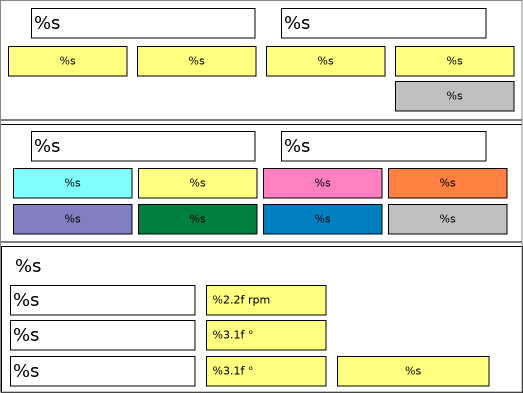
VISUALIZATION VISU_AXE_STD1_LIN_ROT_FCT_CONS_OSC  // 523x393
VAR_IN_OUT
	m_Input_MOTEUR: BLOCK_AXE_STD1_OSCILLANT;
	m_Input_PRG_MOUVEMENT_PS: BLOCK_PRG_MOUVEMENT_PS;
END_VAR
VAR_INPUT CONSTANT
	m_Input_INDEX_MOTEUR : INT;
END_VAR
    Rectangle (0,0 522x120)
    RoundedRectangle (31,8 224x30), "%s", text list: 'TextList_Moteurs', text index: 13
    RoundedRectangle (281,8 205x30), "%s", text variable: m_Input_MOTEUR.CONF_ID_Poste[m_Input_MOTEUR.PRM_NPoste]
    RoundedRectangle (8,46 119x30), "%s", text variable: m_Input_MOTEUR.CONF_ID_Poste[1], invisible if: m_Input_PRG_MOUVEMENT_PS.CONF_NB_POSTE[m_Input_INDEX_MOTEUR]<1, input disabled if: (NOT PRG_User.ACTU_USER.MAINTENANCE AND m_Input_MOTEUR.MANUAL) OR (NOT PRG_User.ACTU_USER.FONCTION_SA AND NOT m_Input_MOTEUR.MANUAL)
        OnMouseClick: execute { m_Input_MOTEUR.PRM_NPOSTE:=1; }
    RoundedRectangle (395,81 119x30), "%s", text variable: m_Input_MOTEUR.CONF_ID_POSTE[0], invisible if: NOT m_Input_PRG_MOUVEMENT_PS.CONF_Use_Poste0[m_Input_INDEX_MOTEUR], input disabled if: (NOT PRG_User.ACTU_USER.MAINTENANCE AND m_Input_MOTEUR.MANUAL) OR (NOT PRG_User.ACTU_USER.FONCTION_SA AND NOT m_Input_MOTEUR.MANUAL)
        OnMouseClick: execute { m_Input_MOTEUR.PRM_NPOSTE:=0; }
    RoundedRectangle (137,46 119x30), "%s", text variable: m_Input_MOTEUR.CONF_ID_Poste[2], invisible if: m_Input_PRG_MOUVEMENT_PS.CONF_NB_POSTE[m_Input_INDEX_MOTEUR]<2, input disabled if: (NOT PRG_User.ACTU_USER.MAINTENANCE AND m_Input_MOTEUR.MANUAL) OR (NOT PRG_User.ACTU_USER.FONCTION_SA AND NOT m_Input_MOTEUR.MANUAL)
        OnMouseClick: execute { m_Input_MOTEUR.PRM_NPOSTE:=2; }
    RoundedRectangle (266,46 119x30), "%s", text variable: m_Input_MOTEUR.CONF_ID_Poste[3], invisible if: m_Input_PRG_MOUVEMENT_PS.CONF_NB_POSTE[m_Input_INDEX_MOTEUR]<3, input disabled if: (NOT PRG_User.ACTU_USER.MAINTENANCE AND m_Input_MOTEUR.MANUAL) OR (NOT PRG_User.ACTU_USER.FONCTION_SA AND NOT m_Input_MOTEUR.MANUAL)
        OnMouseClick: execute { m_Input_MOTEUR.PRM_NPOSTE:=3; }
    RoundedRectangle (395,46 119x30), "%s", text variable: m_Input_MOTEUR.CONF_ID_Poste[4], invisible if: m_Input_PRG_MOUVEMENT_PS.CONF_NB_POSTE[m_Input_INDEX_MOTEUR]<4, input disabled if: (NOT PRG_User.ACTU_USER.MAINTENANCE AND m_Input_MOTEUR.MANUAL) OR (NOT PRG_User.ACTU_USER.FONCTION_SA AND NOT m_Input_MOTEUR.MANUAL)
        OnMouseClick: execute { m_Input_MOTEUR.PRM_NPOSTE:=4; }
    Rectangle (0,124 522x118)
    RoundedRectangle (31,131 224x30), "%s", text list: 'TextList_Moteurs', text index: 14
    RoundedRectangle (281,131 205x30), "%s", text variable: m_Input_MOTEUR.CONF_ID_Ref[m_Input_MOTEUR.PRM_NRef]
    RoundedRectangle (13,168 119x30), "%s", text variable: m_Input_MOTEUR.CONF_ID_REF[1], invisible if: m_Input_PRG_MOUVEMENT_PS.CONF_NB_REF[m_Input_INDEX_MOTEUR]<1, input disabled if: (NOT PRG_User.ACTU_USER.MAINTENANCE AND m_Input_MOTEUR.MANUAL) OR (NOT PRG_User.ACTU_USER.FONCTION_SA AND NOT m_Input_MOTEUR.MANUAL)
        OnMouseClick: execute { m_Input_MOTEUR.PRM_NREF:=1; }
    RoundedRectangle (138,168 119x30), "%s", text variable: m_Input_MOTEUR.CONF_ID_REF[2], invisible if: m_Input_PRG_MOUVEMENT_PS.CONF_NB_REF[m_Input_INDEX_MOTEUR]<2, input disabled if: (NOT PRG_User.ACTU_USER.MAINTENANCE AND m_Input_MOTEUR.MANUAL) OR (NOT PRG_User.ACTU_USER.FONCTION_SA AND NOT m_Input_MOTEUR.MANUAL)
        OnMouseClick: execute { m_Input_MOTEUR.PRM_NREF:=2; }
    RoundedRectangle (263,168 119x30), "%s", text variable: m_Input_MOTEUR.CONF_ID_REF[3], invisible if: m_Input_PRG_MOUVEMENT_PS.CONF_NB_REF[m_Input_INDEX_MOTEUR]<3, input disabled if: (NOT PRG_User.ACTU_USER.MAINTENANCE AND m_Input_MOTEUR.MANUAL) OR (NOT PRG_User.ACTU_USER.FONCTION_SA AND NOT m_Input_MOTEUR.MANUAL)
        OnMouseUp: execute { m_Input_MOTEUR.PRM_NREF:=3; }
    RoundedRectangle (388,168 119x30), "%s", text variable: m_Input_MOTEUR.CONF_ID_REF[4], invisible if: m_Input_PRG_MOUVEMENT_PS.CONF_NB_REF[m_Input_INDEX_MOTEUR]<4, input disabled if: (NOT PRG_User.ACTU_USER.MAINTENANCE AND m_Input_MOTEUR.MANUAL) OR (NOT PRG_User.ACTU_USER.FONCTION_SA AND NOT m_Input_MOTEUR.MANUAL)
        OnMouseClick: execute { m_Input_MOTEUR.PRM_NREF:=4; }
    RoundedRectangle (13,204 119x30), "%s", text variable: m_Input_MOTEUR.CONF_ID_REF[5], invisible if: m_Input_PRG_MOUVEMENT_PS.CONF_NB_REF[m_Input_INDEX_MOTEUR]<5, input disabled if: (NOT PRG_User.ACTU_USER.MAINTENANCE AND m_Input_MOTEUR.MANUAL) OR (NOT PRG_User.ACTU_USER.FONCTION_SA AND NOT m_Input_MOTEUR.MANUAL)
        OnMouseClick: execute { m_Input_MOTEUR.PRM_NREF:=5; }
    RoundedRectangle (138,204 119x30), "%s", text variable: m_Input_MOTEUR.CONF_ID_REF[6], invisible if: m_Input_PRG_MOUVEMENT_PS.CONF_NB_REF[m_Input_INDEX_MOTEUR]<6, input disabled if: (NOT PRG_User.ACTU_USER.MAINTENANCE AND m_Input_MOTEUR.MANUAL) OR (NOT PRG_User.ACTU_USER.FONCTION_SA AND NOT m_Input_MOTEUR.MANUAL)
        OnMouseClick: execute { m_Input_MOTEUR.PRM_NREF:=6; }
    RoundedRectangle (388,204 119x30), "%s", text variable: m_Input_MOTEUR.CONF_ID_REF[0], invisible if: NOT m_Input_PRG_MOUVEMENT_PS.CONF_Use_Ref0[m_Input_INDEX_MOTEUR], input disabled if: (NOT PRG_User.ACTU_USER.MAINTENANCE AND m_Input_MOTEUR.MANUAL) OR (NOT PRG_User.ACTU_USER.FONCTION_SA AND NOT m_Input_MOTEUR.MANUAL)
        OnMouseClick: execute { m_Input_MOTEUR.PRM_NREF:=0; }
    RoundedRectangle (263,204 119x30), "%s", text variable: m_Input_MOTEUR.CONF_ID_REF[7], invisible if: m_Input_PRG_MOUVEMENT_PS.CONF_NB_REF[m_Input_INDEX_MOTEUR]<7, input disabled if: (NOT PRG_User.ACTU_USER.MAINTENANCE AND m_Input_MOTEUR.MANUAL) OR (NOT PRG_User.ACTU_USER.FONCTION_SA AND NOT m_Input_MOTEUR.MANUAL)
        OnMouseClick: execute { m_Input_MOTEUR.PRM_NREF:=7; }
    Rectangle (1,246 522x147)
    RoundedRectangle (10,320 185x30), "%s", invisible if: NOT m_Input_PRG_MOUVEMENT_PS.CONF_Balayage[m_Input_INDEX_MOTEUR] AND NOT m_Input_PRG_MOUVEMENT_PS.CONF_Positionnement[m_Input_INDEX_MOTEUR], text list: 'TextList_Moteurs', text index: 12
    RoundedRectangle (206,320 120x30), "%3.1f mm", text variable: m_Input_MOTEUR.PRM_Position, invisible if: (NOT m_Input_PRG_MOUVEMENT_PS.CONF_Balayage[m_Input_INDEX_MOTEUR] AND NOT m_Input_PRG_MOUVEMENT_PS.CONF_Positionnement[m_Input_INDEX_MOTEUR]) OR NOT m_Input_MOTEUR.CONF_Mvt_Lineaire, input disabled if: (NOT PRG_User.ACTU_USER.MAINTENANCE AND m_Input_MOTEUR.MANUAL) OR (NOT PRG_User.ACTU_USER.FONCTION_SA AND NOT m_Input_MOTEUR.MANUAL)
        OnMouseClick: write the text variable via VisuDialogs.Numpad, min m_Input_PRG_MOUVEMENT_PS.CONF_MIN_POS[m_Input_INDEX_MOTEUR], max m_Input_PRG_MOUVEMENT_PS.CONF_MAX_POS[m_Input_INDEX_MOTEUR]
    RoundedRectangle (10,285 185x30), "%s", invisible if: NOT m_Input_PRG_MOUVEMENT_PS.CONF_Balayage[m_Input_INDEX_MOTEUR] AND NOT m_Input_PRG_MOUVEMENT_PS.CONF_Rotation[m_Input_INDEX_MOTEUR], text list: 'TextList_Moteurs', text index: 7
    RoundedRectangle (206,285 120x30), "%2.2f mmps", text variable: m_Input_MOTEUR.PRM_V_BalRot, invisible if: (NOT m_Input_PRG_MOUVEMENT_PS.CONF_Balayage[m_Input_INDEX_MOTEUR] AND NOT m_Input_PRG_MOUVEMENT_PS.CONF_Rotation[m_Input_INDEX_MOTEUR]) OR NOT m_Input_MOTEUR.CONF_Mvt_Lineaire, input disabled if: (NOT PRG_User.ACTU_USER.MAINTENANCE AND m_Input_MOTEUR.MANUAL) OR (NOT PRG_User.ACTU_USER.FONCTION_SA AND NOT m_Input_MOTEUR.MANUAL)
        OnMouseClick: write the text variable via VisuDialogs.Numpad, min m_Input_PRG_MOUVEMENT_PS.CONF_MIN_SPEED[m_Input_INDEX_MOTEUR], max m_Input_PRG_MOUVEMENT_PS.CONF_MAX_SPEED[m_Input_INDEX_MOTEUR]
    RoundedRectangle (10,356 185x30), "%s", invisible if: NOT m_Input_PRG_MOUVEMENT_PS.CONF_Balayage[m_Input_INDEX_MOTEUR], text list: 'TextList_Moteurs', text index: 16
    RoundedRectangle (206,356 120x30), "%3.1f mm", text variable: m_Input_MOTEUR.PRM_Angle_Bal, invisible if: NOT m_Input_PRG_MOUVEMENT_PS.CONF_Balayage[m_Input_INDEX_MOTEUR] OR NOT m_Input_MOTEUR.CONF_Mvt_Lineaire, input disabled if: (NOT PRG_User.ACTU_USER.MAINTENANCE AND m_Input_MOTEUR.MANUAL) OR (NOT PRG_User.ACTU_USER.FONCTION_SA AND NOT m_Input_MOTEUR.MANUAL)
        OnMouseClick: write the text variable via VisuDialogs.Numpad
    RoundedRectangle (337,356 152x30), "%s", invisible if: NOT m_Input_PRG_MOUVEMENT_PS.CONF_Balayage[m_Input_INDEX_MOTEUR] OR NOT m_Input_MOTEUR.PRM_BalPos, input disabled if: (NOT PRG_User.ACTU_USER.MAINTENANCE AND m_Input_MOTEUR.MANUAL) OR (NOT PRG_User.ACTU_USER.FONCTION_SA AND NOT m_Input_MOTEUR.MANUAL), text list: 'TextList_Moteurs', text index: 21
        toggle m_Input_MOTEUR.PRM_BalPos
    RoundedRectangle (337,356 152x30), "%s", invisible if: NOT m_Input_PRG_MOUVEMENT_PS.CONF_Balayage[m_Input_INDEX_MOTEUR] OR m_Input_MOTEUR.PRM_BalPos, input disabled if: (NOT PRG_User.ACTU_USER.MAINTENANCE AND m_Input_MOTEUR.MANUAL) OR (NOT PRG_User.ACTU_USER.FONCTION_SA AND NOT m_Input_MOTEUR.MANUAL), text list: 'TextList_Process', text index: 22
        toggle m_Input_MOTEUR.PRM_BalPos
    RoundedRectangle (12,251 390x30), "%s", text list: 'TextList_Moteurs', text index: 15
    RoundedRectangle (206,285 120x30), "%2.2f rpm", text variable: m_Input_MOTEUR.PRM_V_BalRot, invisible if: (NOT m_Input_PRG_MOUVEMENT_PS.CONF_Balayage[m_Input_INDEX_MOTEUR] AND NOT m_Input_PRG_MOUVEMENT_PS.CONF_Rotation[m_Input_INDEX_MOTEUR]) OR m_Input_MOTEUR.CONF_Mvt_Lineaire, input disabled if: (NOT PRG_User.ACTU_USER.MAINTENANCE AND m_Input_MOTEUR.MANUAL) OR (NOT PRG_User.ACTU_USER.FONCTION_SA AND NOT m_Input_MOTEUR.MANUAL)
        OnMouseClick: write the text variable via VisuDialogs.Numpad, min m_Input_PRG_MOUVEMENT_PS.CONF_MIN_SPEED[m_Input_INDEX_MOTEUR], max m_Input_PRG_MOUVEMENT_PS.CONF_MAX_SPEED[m_Input_INDEX_MOTEUR]
    RoundedRectangle (206,320 120x30), "%3.1f °", text variable: m_Input_MOTEUR.PRM_Position, invisible if: (NOT m_Input_PRG_MOUVEMENT_PS.CONF_Balayage[m_Input_INDEX_MOTEUR] AND NOT m_Input_PRG_MOUVEMENT_PS.CONF_Positionnement[m_Input_INDEX_MOTEUR]) OR m_Input_MOTEUR.CONF_Mvt_Lineaire, input disabled if: (NOT PRG_User.ACTU_USER.MAINTENANCE AND m_Input_MOTEUR.MANUAL) OR (NOT PRG_User.ACTU_USER.FONCTION_SA AND NOT m_Input_MOTEUR.MANUAL)
        OnMouseClick: write the text variable via VisuDialogs.Numpad, min m_Input_PRG_MOUVEMENT_PS.CONF_MIN_POS[m_Input_INDEX_MOTEUR], max m_Input_PRG_MOUVEMENT_PS.CONF_MAX_POS[m_Input_INDEX_MOTEUR]
    RoundedRectangle (206,356 120x30), "%3.1f °", text variable: m_Input_MOTEUR.PRM_Angle_Bal, invisible if: NOT m_Input_PRG_MOUVEMENT_PS.CONF_Balayage[m_Input_INDEX_MOTEUR] OR m_Input_MOTEUR.CONF_Mvt_Lineaire, input disabled if: (NOT PRG_User.ACTU_USER.MAINTENANCE AND m_Input_MOTEUR.MANUAL) OR (NOT PRG_User.ACTU_USER.FONCTION_SA AND NOT m_Input_MOTEUR.MANUAL)
        OnMouseClick: write the text variable via VisuDialogs.Numpad, min 0, max 360
END_VISUALIZATION

(* stored: Version 1.1.0.1, ProductVersion 3.1.4024.10
   Visu VISU_AXE_STD1_LIN_ROT_FCT_CONS_OSC: Id {bbe0efe5-4fb3-4f59-9dc2-f2245c75d03f} *)
